KUKA KRL program: wkz2_off_stb_ltb.src, wkz2_off_stb_ltb.dat

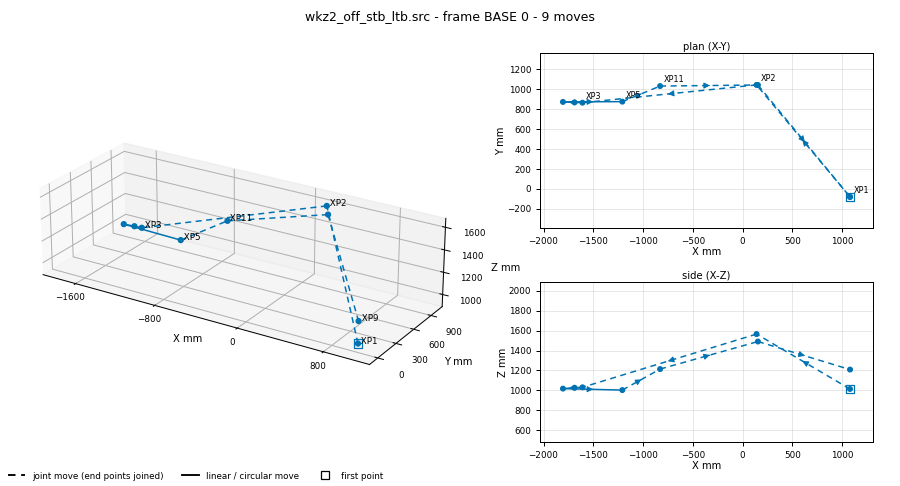
[picture p0: tool path of wkz2_off_stb_ltb.src in frame BASE 0, 9 of 9 moves have a stored position in this frame; points joined in program order, loops and branches not executed]
--- wkz2_off_stb_ltb.src ---
&ACCESS RV1
&REL 13
&PARAM DISKPATH = Program/WKZ
DEF wkz2_off_stb_ltb( )
;FOLD INI
  ;FOLD BASISTECH INI
    GLOBAL INTERRUPT DECL 3 WHEN $STOPMESS==TRUE DO IR_STOPM ( )
    INTERRUPT ON 3
    BAS (#INITMOV,0 )
  ;ENDFOLD (BASISTECH INI)
  ;FOLD USER INI
    ;Make your modifications here
  ;ENDFOLD (USER INI)
;ENDFOLD (INI)

; Caracterização dos meios de produção:
; Versão Atual:
; 04/05/2013 12:00 Name: P13.090-R6 CHANGES: Posicionamento de garra Actros
; para geometria
$ov_pro=50
chk_w2_wechs_ok ( )  ; VERIFICAÇÃO DE FERRAMENTA: GRIPPER ACTROS

;FOLD PTP P1 Vel=50 % PDAT1 Tool[2]:Gripper Parabrisa Actro Base[0];%{PE}%R 8.2.24,%MKUKATPBASIS,%CMOVE,%VPTP,%P 1:PTP, 2:P1, 3:, 5:50, 7:PDAT1
$BWDSTART=FALSE
PDAT_ACT=PPDAT1
FDAT_ACT=FP1
BAS(#PTP_PARAMS,50)
PTP XP1
;ENDFOLD

;FOLD ; SET GRAMPOS 1 a 4 OPEN;%{PE}%R 8.2.24,%MKUKATPBASIS,%CCOMMENT,%VNORMAL,%P 2:SET  GRAMPOS  1  a  4  OPEN
;ENDFOLD
;FOLD SET GRP 1 State=OPN GDAT1;%{PE}%R 8.2.4,%MKUKATPGRP,%CGRP,%VGRP,%P 2:1, 4:2, 5:#NO, 6:GDAT1, 8:0, 10:0
H50(GRP,1,2,GGDAT1)
;ENDFOLD
;FOLD SET GRP 2 State=OPN GDAT2;%{PE}%R 8.2.4,%MKUKATPGRP,%CGRP,%VGRP,%P 2:2, 4:2, 5:#NO, 6:GDAT2, 8:0, 10:0
H50(GRP,2,2,GGDAT2)
;ENDFOLD
;FOLD SET GRP 3 State=OPN GDAT3;%{PE}%R 8.2.4,%MKUKATPGRP,%CGRP,%VGRP,%P 2:3, 4:2, 5:#NO, 6:GDAT3, 8:0, 10:0
H50(GRP,3,2,GGDAT3)
;ENDFOLD
;FOLD SET GRP 4 State=OPN GDAT9;%{PE}%R 8.2.4,%MKUKATPGRP,%CGRP,%VGRP,%P 2:4, 4:2, 5:#NO, 6:GDAT9, 8:0, 10:0
H50(GRP,4,2,GGDAT9)
;ENDFOLD

;FOLD ; CHECAR SE GRUPOS DE GRAMPOS 1 a 4 ESTAO ABERTOS;%{PE}%R 8.2.24,%MKUKATPBASIS,%CCOMMENT,%VNORMAL,%P 2:CHECAR  SE  GRUPOS  DE  GRAMPOS  1  a  4  ESTAO  ABERTOS
;ENDFOLD
chk_w2_grp1_opn ()
chk_w2_grp2_opn ()
chk_w2_grp3_opn ()
chk_w2_grp4_opn ()

;FOLD WAIT FOR ( IN 3340 'AGUARDA LIB FAZER GEOMETRIA' );%{PE}%R 8.2.24,%MKUKATPBASIS,%CEXT_WAIT_FOR,%VEXT_WAIT_FOR,%P 2:, 4:, 5:$IN, 6:3340, 7:AGUARDA LIB FAZER GEOMETRIA, 9:
WAIT FOR  ( $IN[3340] )
;ENDFOLD
;FOLD OUT 3321 'FORA DA GEOMETRIA' State=TRUE ;%{PE}%R 8.2.24,%MKUKATPBASIS,%COUT,%VOUTX,%P 2:3321, 3:FORA DA GEOMETRIA, 5:TRUE, 6:
$OUT[3321]=TRUE
;ENDFOLD

;FOLD PTP P2 CONT Vel=50 % PDAT2 Tool[2]:Gripper Parabrisa Actro Base[0];%{PE}%R 8.2.24,%MKUKATPBASIS,%CMOVE,%VPTP,%P 1:PTP, 2:P2, 3:C_PTP, 5:50, 7:PDAT2
$BWDSTART=FALSE
PDAT_ACT=PPDAT2
FDAT_ACT=FP2
BAS(#PTP_PARAMS,50)
PTP XP2 C_PTP
;ENDFOLD
;FOLD PTP P3 Vel=50 % PDAT3 Tool[2]:Gripper Parabrisa Actro Base[0];%{PE}%R 8.2.24,%MKUKATPBASIS,%CMOVE,%VPTP,%P 1:PTP, 2:P3, 3:, 5:50, 7:PDAT3
$BWDSTART=FALSE
PDAT_ACT=PPDAT3
FDAT_ACT=FP3
BAS(#PTP_PARAMS,50)
PTP XP3
;ENDFOLD
;FOLD LIN P10 Vel=0.2 m/s CPDAT4 Tool[2]:Gripper Parabrisa Actro Base[0];%{PE}%R 8.2.24,%MKUKATPBASIS,%CMOVE,%VLIN,%P 1:LIN, 2:P10, 3:, 5:0.2, 7:CPDAT4
$BWDSTART=FALSE
LDAT_ACT=LCPDAT4
FDAT_ACT=FP10
BAS(#CP_PARAMS,0.2)
LIN XP10
;ENDFOLD

;FOLD ; PONTO DE GEOMETRIA;%{PE}%R 8.2.24,%MKUKATPBASIS,%CCOMMENT,%VNORMAL,%P 2:PONTO  DE  GEOMETRIA
;ENDFOLD
;FOLD LIN P4 Vel=0.2 m/s CPDAT1 Tool[2]:Gripper Parabrisa Actro Base[0];%{PE}%R 8.2.24,%MKUKATPBASIS,%CMOVE,%VLIN,%P 1:LIN, 2:P4, 3:, 5:0.2, 7:CPDAT1
$BWDSTART=FALSE
LDAT_ACT=LCPDAT1
FDAT_ACT=FP4
BAS(#CP_PARAMS,0.2)
LIN XP4
;ENDFOLD

;FOLD ; FECHAR GRUPOS 1,3 E 2;%{PE}%R 8.2.24,%MKUKATPBASIS,%CCOMMENT,%VNORMAL,%P 2:FECHAR  GRUPOS  1,3  E  2
;ENDFOLD
;FOLD SET GRP 1 State=CLO GDAT4;%{PE}%R 8.2.4,%MKUKATPGRP,%CGRP,%VGRP,%P 2:1, 4:1, 5:#NO, 6:GDAT4, 8:0, 10:0
H50(GRP,1,1,GGDAT4)
;ENDFOLD
chk_w2_grp1_clo ()

;FOLD SET GRP 3 State=CLO GDAT7;%{PE}%R 8.2.4,%MKUKATPGRP,%CGRP,%VGRP,%P 2:3, 4:1, 5:#NO, 6:GDAT7, 8:0, 10:0
H50(GRP,3,1,GGDAT7)
;ENDFOLD
chk_w2_grp3_clo ()

;FOLD SET GRP 2 State=CLO GDAT13;%{PE}%R 8.2.4,%MKUKATPGRP,%CGRP,%VGRP,%P 2:2, 4:1, 5:#NO, 6:GDAT13, 8:0, 10:0
H50(GRP,2,1,GGDAT13)
;ENDFOLD
chk_w2_grp2_clo ()

;FOLD ; Bloco de grampos superiores;%{PE}%R 8.2.24,%MKUKATPBASIS,%CCOMMENT,%VNORMAL,%P 2:Bloco  de  grampos  superiores
;ENDFOLD
;FOLD SET GRP 4 State=CLO GDAT15;%{PE}%R 8.2.4,%MKUKATPGRP,%CGRP,%VGRP,%P 2:4, 4:1, 5:#NO, 6:GDAT15, 8:0, 10:0
H50(GRP,4,1,GGDAT15)
;ENDFOLD
chk_w2_grp4_clo ()

;FOLD OUT 3333 'R6 TRABALHO CONCLUIDO' State=TRUE ;%{PE}%R 8.2.24,%MKUKATPBASIS,%COUT,%VOUTX,%P 2:3333, 3:R6 TRABALHO CONCLUIDO, 5:TRUE, 6:
$OUT[3333]=TRUE
;ENDFOLD
;FOLD OUT 3334 'R6 SOLICITA LIB SAIR' State=TRUE ;%{PE}%R 8.2.24,%MKUKATPBASIS,%COUT,%VOUTX,%P 2:3334, 3:R6 SOLICITA LIB SAIR, 5:TRUE, 6:
$OUT[3334]=TRUE
;ENDFOLD
;FOLD WAIT FOR ( IN 3342 'AGUARDA LIB SAIR COM GARRA' );%{PE}%R 8.2.24,%MKUKATPBASIS,%CEXT_WAIT_FOR,%VEXT_WAIT_FOR,%P 2:, 4:, 5:$IN, 6:3342, 7:AGUARDA LIB SAIR COM GARRA, 9:
WAIT FOR  ( $IN[3342] )
;ENDFOLD
;FOLD OUT 3334 'R6 SOLICITA LIB SAIR' State=FALSE ;%{PE}%R 8.2.24,%MKUKATPBASIS,%COUT,%VOUTX,%P 2:3334, 3:R6 SOLICITA LIB SAIR, 5:FALSE, 6:
$OUT[3334]=FALSE
;ENDFOLD

;FOLD ; ABRIR GRUPOS 1,3 ,4,2;%{PE}%R 8.2.24,%MKUKATPBASIS,%CCOMMENT,%VNORMAL,%P 2:ABRIR  GRUPOS  1,3 ,4,2
;ENDFOLD
;FOLD SET GRP 1 State=OPN GDAT10;%{PE}%R 8.2.4,%MKUKATPGRP,%CGRP,%VGRP,%P 2:1, 4:2, 5:#NO, 6:GDAT10, 8:0, 10:0
H50(GRP,1,2,GGDAT10)
;ENDFOLD
chk_w2_grp1_opn ()

;FOLD SET GRP 3 State=OPN GDAT11;%{PE}%R 8.2.4,%MKUKATPGRP,%CGRP,%VGRP,%P 2:3, 4:2, 5:#NO, 6:GDAT11, 8:0, 10:0
H50(GRP,3,2,GGDAT11)
;ENDFOLD
chk_w2_grp3_opn ()

;FOLD SET GRP 4 State=OPN GDAT12;%{PE}%R 8.2.4,%MKUKATPGRP,%CGRP,%VGRP,%P 2:4, 4:2, 5:#NO, 6:GDAT12, 8:0, 10:0
H50(GRP,4,2,GGDAT12)
;ENDFOLD
chk_w2_grp4_opn ()

;FOLD SET GRP 2 State=OPN GDAT16;%{PE}%R 8.2.4,%MKUKATPGRP,%CGRP,%VGRP,%P 2:2, 4:2, 5:#NO, 6:GDAT16, 8:0, 10:0
H50(GRP,2,2,GGDAT16)
;ENDFOLD
chk_w2_grp2_opn ()

;FOLD OUT 3333 'R6 TRABALHO CONCLUIDO' State=FALSE ;%{PE}%R 8.2.24,%MKUKATPBASIS,%COUT,%VOUTX,%P 2:3333, 3:R6 TRABALHO CONCLUIDO, 5:FALSE, 6:
$OUT[3333]=FALSE
;ENDFOLD

;FOLD LIN P5 Vel=0.2 m/s CPDAT2 Tool[2]:Gripper Parabrisa Actro Base[0];%{PE}%R 8.2.24,%MKUKATPBASIS,%CMOVE,%VLIN,%P 1:LIN, 2:P5, 3:, 5:0.2, 7:CPDAT2
$BWDSTART=FALSE
LDAT_ACT=LCPDAT2
FDAT_ACT=FP5
BAS(#CP_PARAMS,0.2)
LIN XP5
;ENDFOLD
;FOLD PTP P11 Vel=100 % PDAT7 Tool[2]:Gripper Parabrisa Actro Base[0];%{PE}%R 8.2.24,%MKUKATPBASIS,%CMOVE,%VPTP,%P 1:PTP, 2:P11, 3:, 5:100, 7:PDAT7
$BWDSTART=FALSE
PDAT_ACT=PPDAT7
FDAT_ACT=FP11
BAS(#PTP_PARAMS,100)
PTP XP11
;ENDFOLD

;FOLD PULSE 3340 'R6 GEOMETRIA OK' State=TRUE Time=3 sec;%{PE}%R 8.2.24,%MKUKATPBASIS,%COUT,%VPULSE,%P 2:3340, 3:R6 GEOMETRIA OK, 5:TRUE, 6:, 8:3
PULSE($OUT[3340], TRUE,3)
;ENDFOLD

;FOLD PTP P6 Vel=50 % PDAT4 Tool[2]:Gripper Parabrisa Actro Base[0];%{PE}%R 8.2.24,%MKUKATPBASIS,%CMOVE,%VPTP,%P 1:PTP, 2:P6, 3:, 5:50, 7:PDAT4
$BWDSTART=FALSE
PDAT_ACT=PPDAT4
FDAT_ACT=FP6
BAS(#PTP_PARAMS,50)
PTP XP6
;ENDFOLD

;FOLD OUT 3321 'FORA DA GEOMETRIA' State=TRUE ;%{PE}%R 8.2.24,%MKUKATPBASIS,%COUT,%VOUTX,%P 2:3321, 3:FORA DA GEOMETRIA, 5:TRUE, 6:
$OUT[3321]=TRUE
;ENDFOLD

;FOLD PTP P9 Vel=50 % PDAT6 Tool[2]:Gripper Parabrisa Actro Base[0];%{PE}%R 8.2.24,%MKUKATPBASIS,%CMOVE,%VPTP,%P 1:PTP, 2:P9, 3:, 5:50, 7:PDAT6
$BWDSTART=FALSE
PDAT_ACT=PPDAT6
FDAT_ACT=FP9
BAS(#PTP_PARAMS,50)
PTP XP9
;ENDFOLD
$ov_pro=100

END

--- wkz2_off_stb_ltb.dat ---
&ACCESS RV1
&REL 13
&PARAM DISKPATH = Program/WKZ
DEFDAT  wkz2_off_stb_ltb
;FOLD EXTERNAL DECLARATIONS;%{PE}%MKUKATPBASIS,%CEXT,%VCOMMON,%P
;FOLD BASISTECH EXT;%{PE}%MKUKATPBASIS,%CEXT,%VEXT,%P
EXT  BAS (BAS_COMMAND  :IN,REAL  :IN )
DECL INT SUCCESS
;ENDFOLD (BASISTECH EXT)
;FOLD USER EXT;%{E}%MKUKATPUSER,%CEXT,%VEXT,%P
;Make your modifications here
;ENDFOLD (USER EXT)
;ENDFOLD (EXTERNAL DECLARATIONS)

;# ============ START PATH : wkz2_off_lta_mgs =============
DECL FDAT Fnew_wkz2_off_lta_mgs_p2={TOOL_NO 2,BASE_NO 0,IPO_FRAME #BASE,POINT2[] " "}
DECL PDAT PP_OLP1={VEL 50.0,ACC 50.0,APO_DIST 0.0}
DECL E6POS Xnew_wkz2_off_lta_mgs_p2={X 75.9020004,Y 1031.19702,Z 1458.79199,A 50.2246017,B -77.8526993,C -150.349106,S 6,T 19}
DECL FDAT Fnew_wkz2_off_lta_mgs_p4={TOOL_NO 2,BASE_NO 0,IPO_FRAME #BASE,POINT2[] " "}
DECL PDAT PP_OLP2={VEL 50.0,ACC 50.0,APO_DIST 0.0}
DECL E6POS Xnew_wkz2_off_lta_mgs_p4={X -1790.73303,Y 871.689026,Z 1022.927,A -10.6128998,B -87.8082962,C 10.7388,S 6,T 19}
DECL FDAT Fnew_wkz2_off_lta_mgs_p1={TOOL_NO 2,BASE_NO 0,IPO_FRAME #BASE,POINT2[] " "}
DECL E6POS Xnew_wkz2_off_lta_mgs_p1={X -1807.55701,Y 874.252014,Z 1019.41699,A -8.5866003,B -87.2934036,C 8.71070004,S 6,T 19}
DECL LDAT LL_OLP1={VEL 0.200000003,ACC 20.0,APO_DIST 100.0,APO_FAC 50.0,ORI_TYP #VAR,CIRC_TYP #BASE,JERK_FAC 50.0}
DECL FDAT Fnew_wkz2_off_lta_mgs_p5={TOOL_NO 2,BASE_NO 0,IPO_FRAME #BASE,POINT2[] " "}
DECL E6POS Xnew_wkz2_off_lta_mgs_p5={X -1225.25806,Y 877.679993,Z 1013.09698,A -10.8899002,B -88.8499985,C 11.0176001,S 6,T 19}
DECL LDAT LL_OLP2={VEL 0.200000003,ACC 40.0,APO_DIST 0.0,APO_FAC 0.0,ORI_TYP #VAR,CIRC_TYP #BASE,JERK_FAC 50.0}
DECL FDAT Fnew_wkz2_off_lta_mgs_p7={TOOL_NO 2,BASE_NO 0,IPO_FRAME #BASE,POINT2[] " "}
DECL PDAT PP_OLP3={VEL 50.0,ACC 50.0,APO_DIST 0.0}
DECL E6POS Xnew_wkz2_off_lta_mgs_p7={X 75.8949966,Y 1031.19397,Z 1458.78894,A 50.2229996,B -77.8520966,C -150.347305,S 6,T 19}
DECL BASIS_SUGG_T LAST_BASIS={POINT1[] "P11                     ",POINT2[] "P11                     ",CP_PARAMS[] "CPDAT4                  ",PTP_PARAMS[] "PDAT7                   ",CONT[] "                        ",CP_VEL[] "0.2                     ",PTP_VEL[] "100                     ",SYNC_PARAMS[] "SYNCDAT                 ",SPL_NAME[] "S0                      "}
DECL E6POS XP1={X 1078.36694,Y -79.8197479,Z 1013.849,A 0.511396885,B -24.8505898,C 145.9991,S 18,T 2,E1 0.0,E2 0.0,E3 0.0,E4 0.0,E5 0.0,E6 0.0}
DECL FDAT FP1={TOOL_NO 2,BASE_NO 0,IPO_FRAME #BASE,POINT2[] " ",TQ_STATE FALSE}
DECL PDAT PPDAT1={VEL 100.0,ACC 100.0,APO_DIST 100.0,GEAR_JERK 50.0}
DECL E6POS XP2={X 139.7612,Y 1045.13794,Z 1565.71497,A 68.6732635,B -80.8302536,C -169.097595,S 22,T 19,E1 0.0,E2 0.0,E3 0.0,E4 0.0,E5 0.0,E6 0.0}
DECL FDAT FP2={TOOL_NO 2,BASE_NO 0,IPO_FRAME #BASE,POINT2[] " ",TQ_STATE FALSE}
DECL PDAT PPDAT2={VEL 100.0,ACC 100.0,APO_DIST 100.0,APO_MODE #CPTP,GEAR_JERK 50.0}
DECL E6POS XP3={X -1608.54602,Y 866.486877,Z 1030.995,A -8.15907955,B -87.9976425,C 8.41612053,S 22,T 19,E1 0.0,E2 0.0,E3 0.0,E4 0.0,E5 0.0,E6 0.0}
DECL FDAT FP3={TOOL_NO 2,BASE_NO 0,IPO_FRAME #BASE,POINT2[] " ",TQ_STATE FALSE}
DECL PDAT PPDAT3={VEL 100.0,ACC 50.0,APO_DIST 100.0,GEAR_JERK 50.0}
DECL E6POS XP4={X -1804.66003,Y 874.285522,Z 1017.73297,A -3.80735111,B -87.5602036,C 4.00769281,S 22,T 19,E1 0.0,E2 0.0,E3 0.0,E4 0.0,E5 0.0,E6 0.0}
DECL FDAT FP4={TOOL_NO 2,BASE_NO 0,IPO_FRAME #BASE,POINT2[] " ",TQ_STATE FALSE}
DECL LDAT LCPDAT1={VEL 2.0,ACC 40.0,APO_DIST 100.0,APO_FAC 50.0,AXIS_VEL 100.0,AXIS_ACC 100.0,ORI_TYP #VAR,CIRC_TYP #BASE,JERK_FAC 50.0,GEAR_JERK 50.0,EXAX_IGN 0}
DECL E6POS XP5={X -1208.396,Y 877.059021,Z 1003.01099,A -2.27772999,B -88.4549179,C 2.55537701,S 22,T 19,E1 0.0,E2 0.0,E3 0.0,E4 0.0,E5 0.0,E6 0.0}
DECL FDAT FP5={TOOL_NO 2,BASE_NO 0,IPO_FRAME #BASE,POINT2[] " ",TQ_STATE FALSE}
DECL LDAT LCPDAT2={VEL 2.0,ACC 20.0,APO_DIST 100.0,APO_FAC 50.0,AXIS_VEL 100.0,AXIS_ACC 100.0,ORI_TYP #VAR,CIRC_TYP #BASE,JERK_FAC 50.0,GEAR_JERK 50.0,EXAX_IGN 0}
DECL E6POS XP6={X 153.680695,Y 1044.38306,Z 1490.76099,A 76.7332306,B -81.4597015,C -177.251999,S 22,T 19,E1 0.0,E2 0.0,E3 0.0,E4 0.0,E5 0.0,E6 0.0}
DECL FDAT FP6={TOOL_NO 2,BASE_NO 0,IPO_FRAME #BASE,POINT2[] " ",TQ_STATE FALSE}
DECL PDAT PPDAT4={VEL 100.0,ACC 50.0,APO_DIST 100.0,APO_MODE #CPTP,GEAR_JERK 50.0}
DECL GRP_SUGG_T LAST_GRP={NUMBER[] "2                       ",STATE[] "2                       ",PARAMS[] "GDAT16                  "}
DECL GRP_TYP GCONT={G_APO #YES,GRP_TIME 0.0,CTRL #OFF,DLY 0,DST 0}
DECL E6POS XP7={X -1208.19897,Y 877.023621,Z 1002.60199,A -2.82440495,B -88.4650497,C 3.1100409,S 22,T 19,E1 0.0,E2 0.0,E3 0.0,E4 0.0,E5 0.0,E6 0.0}
DECL FDAT FP7={TOOL_NO 2,BASE_NO 0,IPO_FRAME #BASE,POINT2[] " ",TQ_STATE FALSE}
DECL LDAT LCPDAT3={VEL 2.0,ACC 40.0,APO_DIST 100.0,APO_FAC 50.0,AXIS_VEL 100.0,AXIS_ACC 100.0,ORI_TYP #VAR,CIRC_TYP #BASE,JERK_FAC 50.0,GEAR_JERK 50.0,EXAX_IGN 0}
DECL E6POS XP8={X 1078.45801,Y -79.6040421,Z 954.659973,A 0.500513792,B -24.8502007,C 146.010895,S 18,T 2,E1 0.0,E2 0.0,E3 0.0,E4 0.0,E5 0.0,E6 0.0}
DECL FDAT FP8={TOOL_NO 2,BASE_NO 0,IPO_FRAME #BASE,POINT2[] " ",TQ_STATE FALSE}
DECL PDAT PPDAT5={VEL 100.0,ACC 100.0,APO_DIST 100.0,GEAR_JERK 50.0}
DECL PDAT PPDAT6={VEL 100.0,ACC 100.0,APO_DIST 100.0,GEAR_JERK 50.0}
DECL E6POS XP9={X 1078.83105,Y -80.4085693,Z 1209.02905,A 0.508503377,B -24.8566895,C 145.988495,S 18,T 2,E1 0.0,E2 0.0,E3 0.0,E4 0.0,E5 0.0,E6 0.0}
DECL FDAT FP9={TOOL_NO 2,BASE_NO 0,IPO_FRAME #BASE,POINT2[] " ",TQ_STATE FALSE}
DECL GRP_TYP GGDAT1={G_APO #NO,GRP_TIME 0.200000003,CTRL #OFF,DLY 0,DST 1}
DECL GRP_TYP GGDAT2={G_APO #NO,GRP_TIME 0.200000003,CTRL #OFF,DLY 0,DST 1}
DECL GRP_TYP GGDAT3={G_APO #NO,GRP_TIME 0.200000003,CTRL #OFF,DLY 0,DST 1}
DECL GRP_TYP GGDAT9={G_APO #NO,GRP_TIME 0.200000003,CTRL #OFF,DLY 0,DST 1}
DECL GRP_TYP GGDAT4={G_APO #NO,GRP_TIME 0.200000003,CTRL #OFF,DLY 0,DST 1}
DECL GRP_TYP GGDAT5={G_APO #NO,GRP_TIME 0.200000003,CTRL #OFF,DLY 0,DST 1}
DECL GRP_TYP GGDAT6={G_APO #NO,GRP_TIME 0.200000003,CTRL #OFF,DLY 0,DST 1}
DECL GRP_TYP GGDAT7={G_APO #NO,GRP_TIME 0.200000003,CTRL #OFF,DLY 0,DST 1}
DECL GRP_TYP GGDAT8={G_APO #NO,GRP_TIME 0.200000003,CTRL #OFF,DLY 0,DST 1}
DECL GRP_TYP GGDAT10={G_APO #NO,GRP_TIME 0.200000003,CTRL #OFF,DLY 0,DST 1}
DECL GRP_TYP GGDAT11={G_APO #NO,GRP_TIME 0.200000003,CTRL #OFF,DLY 0,DST 1}
DECL GRP_TYP GGDAT12={G_APO #NO,GRP_TIME 0.200000003,CTRL #OFF,DLY 0,DST 1}
DECL E6POS XP10={X -1687.90503,Y 869.543579,Z 1026.12097,A -6.44977713,B -88.1939468,C 6.72676182,S 22,T 19,E1 0.0,E2 0.0,E3 0.0,E4 0.0,E5 0.0,E6 0.0}
DECL FDAT FP10={TOOL_NO 2,BASE_NO 0,IPO_FRAME #BASE,POINT2[] " ",TQ_STATE FALSE}
DECL LDAT LCPDAT4={VEL 2.0,ACC 100.0,APO_DIST 100.0,APO_FAC 50.0,AXIS_VEL 100.0,AXIS_ACC 100.0,ORI_TYP #VAR,CIRC_TYP #BASE,JERK_FAC 50.0,GEAR_JERK 50.0,EXAX_IGN 0}
DECL E6POS XP11={X -829.034912,Y 1033.58105,Z 1213.97705,A 97.0139771,B -87.2552567,C -115.695602,S 22,T 19,E1 0.0,E2 0.0,E3 0.0,E4 0.0,E5 0.0,E6 0.0}
DECL FDAT FP11={TOOL_NO 2,BASE_NO 0,IPO_FRAME #BASE,POINT2[] " ",TQ_STATE FALSE}
DECL PDAT PPDAT7={VEL 100.0,ACC 100.0,APO_DIST 100.0,GEAR_JERK 50.0}
DECL GRP_TYP GGDAT13={G_APO #NO,GRP_TIME 0.200000003,CTRL #OFF,DLY 0,DST 1}
DECL GRP_TYP GGDAT14={G_APO #NO,GRP_TIME 0.200000003,CTRL #OFF,DLY 0,DST 1}
DECL GRP_TYP GGDAT15={G_APO #NO,GRP_TIME 0.200000003,CTRL #OFF,DLY 0,DST 1}
DECL GRP_TYP GGDAT16={G_APO #NO,GRP_TIME 0.200000003,CTRL #OFF,DLY 0,DST 1}
ENDDAT
